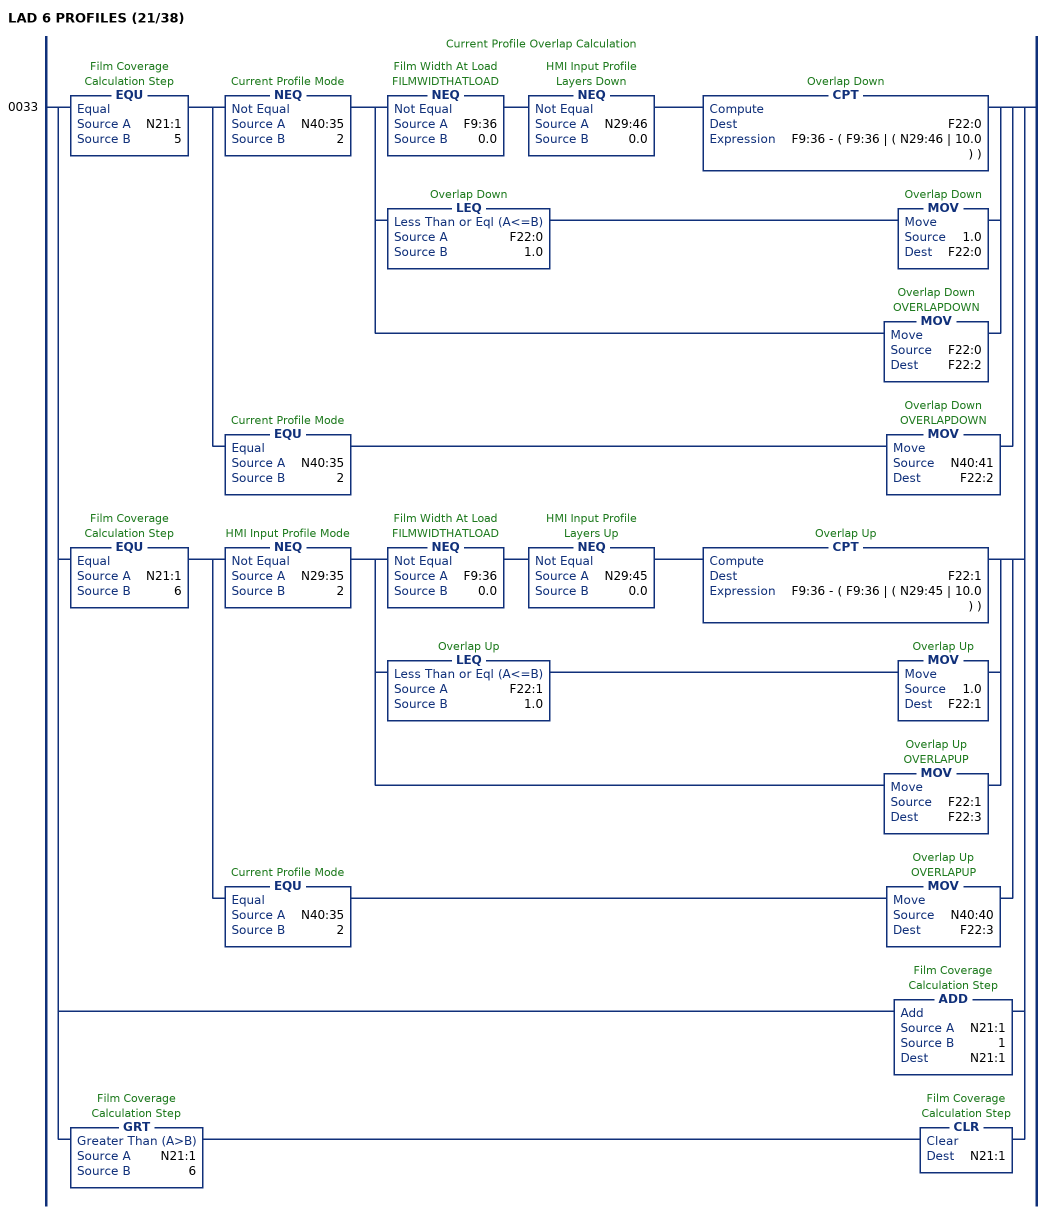
% Rung: 33 %
% Current Profile Overlap Calculation %
SOR BST EQU N21:1 5 BST NEQ N40:35 2 BST NEQ F9:36 0.0 NEQ N29:46 0.0 CPT F22:0 " F9:36 - ( F9:36 | ( N29:46 | 10.0 ) ) " NXB LEQ F22:0 1.0 MOV 1.0 F22:0 NXB MOV F22:0 F22:2 BND NXB EQU N40:35 2 MOV N40:41 F22:2 BND NXB EQU N21:1 6 BST NEQ N29:35 2 BST NEQ F9:36 0.0 NEQ N29:45 0.0 CPT F22:1 " F9:36 - ( F9:36 | ( N29:45 | 10.0 ) ) " NXB LEQ F22:1 1.0 MOV 1.0 F22:1 NXB MOV F22:1 F22:3 BND NXB EQU N40:35 2 MOV N40:40 F22:3 BND NXB BST ADD N21:1 1 N21:1 NXB GRT N21:1 6 CLR N21:1 BND BND EOR
%   N21:1  "Film Coverage Calculation Step" %
%   N40:35  "Current Profile Mode" %
%   F9:36  FILMWIDTHATLOAD  "Film Width At Load" %
%   N29:46  "HMI Input Profile Layers Down" %
%   F22:0  "Overlap Down" %
%   F22:2  OVERLAPDOWN  "Overlap Down" %
%   N29:35  "HMI Input Profile Mode" %
%   N29:45  "HMI Input Profile Layers Up" %
%   F22:1  "Overlap Up" %
%   F22:3  OVERLAPUP  "Overlap Up" %

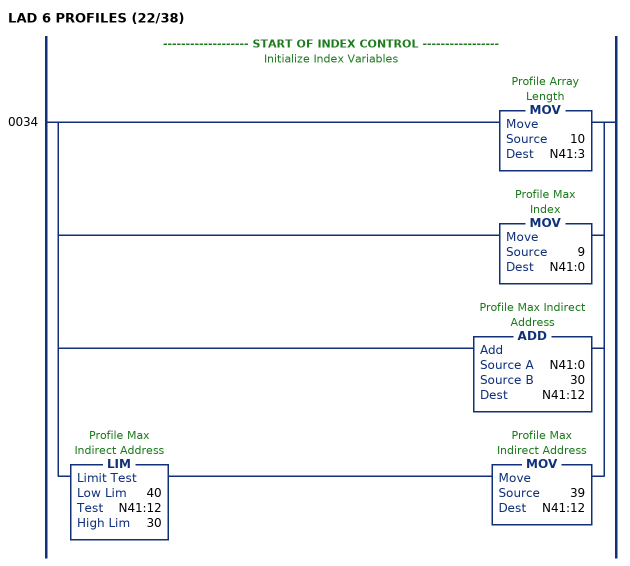
% Rung: 34 %
% TITLE: ------------------- START OF INDEX CONTROL ----------------- %
% Initialize Index Variables %
SOR BST MOV 10 N41:3 NXB MOV 9 N41:0 NXB ADD N41:0 30 N41:12 NXB LIM 40 N41:12 30 MOV 39 N41:12 BND EOR
%   N41:3  "Profile Array Length" %
%   N41:0  "Profile Max Index" %
%   N41:12  "Profile Max Indirect Address" %

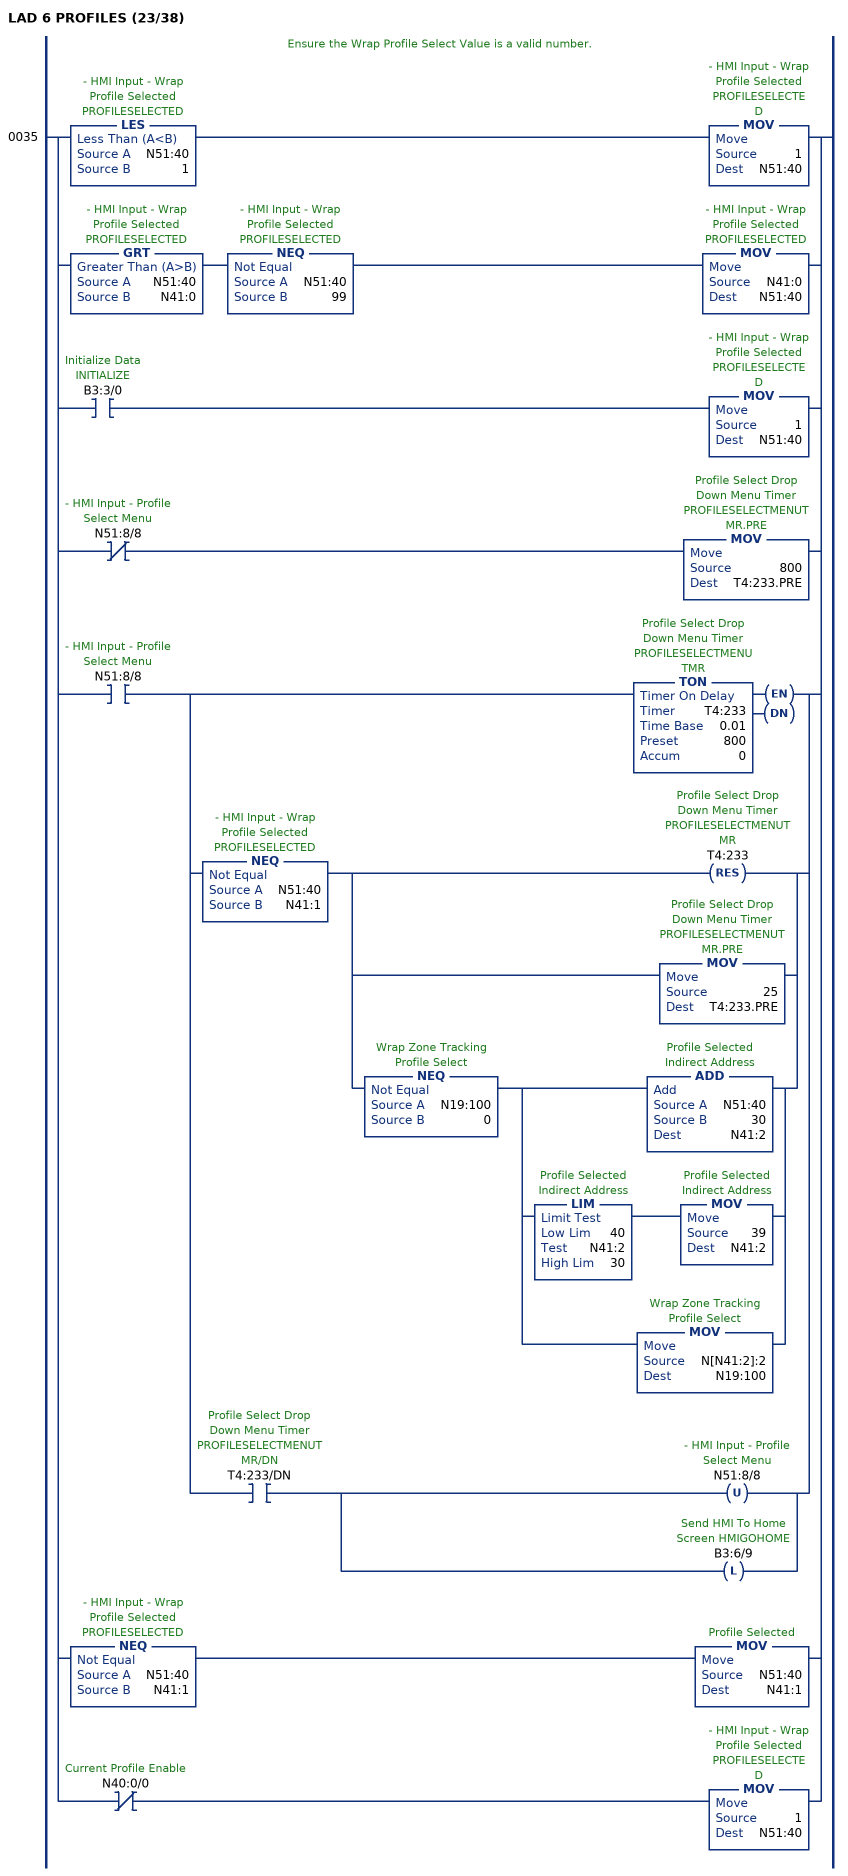
% Rung: 35 %
% Ensure the Wrap Profile Select Value is a valid number. %
SOR BST LES N51:40 1 MOV 1 N51:40 NXB GRT N51:40 N41:0 NEQ N51:40 99 MOV N41:0 N51:40 NXB XIC B3:3/0 MOV 1 N51:40 NXB XIO N51:8/8 MOV 800 T4:233.PRE NXB XIC N51:8/8 BST TON T4:233 0.01 800 0 NXB NEQ N51:40 N41:1 BST RES T4:233 NXB MOV 25 T4:233.PRE NXB NEQ N19:100 0 BST ADD N51:40 30 N41:2 NXB LIM 40 N41:2 30 MOV 39 N41:2 NXB MOV N[N41:2]:2 N19:100 BND BND NXB XIC T4:233/DN BST OTU N51:8/8 NXB OTL B3:6/9 BND BND NXB NEQ N51:40 N41:1 MOV N51:40 N41:1 NXB XIO N40:0/0 MOV 1 N51:40 BND EOR
%   N51:40  PROFILESELECTED  "- HMI Input - Wrap Profile Selected" %
%   N41:0  "Profile Max Index" %
%   B3:3/0  INITIALIZE  "Initialize Data" %
%   N51:8/8  "- HMI Input - Profile Select Menu" %
%   T4:233  PROFILESELECTMENUTMR  "Profile Select Drop Down Menu Timer" %
%   N41:1  "Profile Selected" %
%   N19:100  "Wrap Zone Tracking Profile Select" %
%   N41:2  "Profile Selected Indirect Address" %
%   B3:6/9  HMIGOHOME  "Send HMI To Home Screen" %
%   N40:0/0  "Current Profile Enable" %

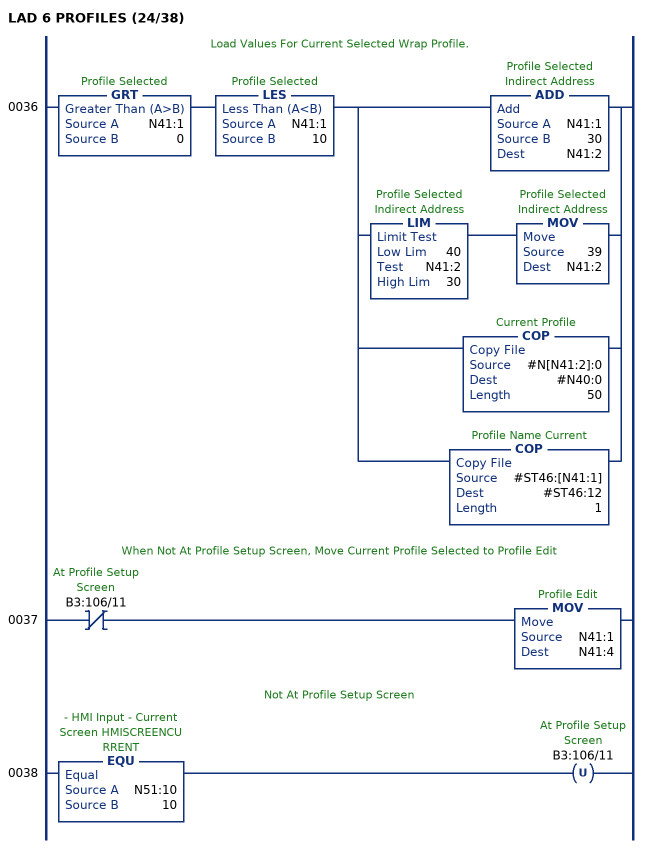
% Rung: 36 %
% Load Values For Current Selected Wrap Profile. %
SOR GRT N41:1 0 LES N41:1 10 BST ADD N41:1 30 N41:2 NXB LIM 40 N41:2 30 MOV 39 N41:2 NXB COP #N[N41:2]:0 #N40:0 50 NXB COP #ST46:[N41:1] #ST46:12 1 BND EOR
%   N41:1  "Profile Selected" %
%   N41:2  "Profile Selected Indirect Address" %
%   N40:0  "Current Profile" %
%   ST46:12  "Profile Name Current" %
% Rung: 37 %
% When Not At Profile Setup Screen, Move Current Profile Selected to Profile Edit %
SOR XIO B3:106/11 MOV N41:1 N41:4 EOR
%   B3:106/11  "At Profile Setup Screen" %
%   N41:1  "Profile Selected" %
%   N41:4  "Profile Edit" %
% Rung: 38 %
% Not At Profile Setup Screen %
SOR EQU N51:10 10 OTU B3:106/11 EOR
%   N51:10  HMISCREENCURRENT  "- HMI Input - Current Screen" %
%   B3:106/11  "At Profile Setup Screen" %

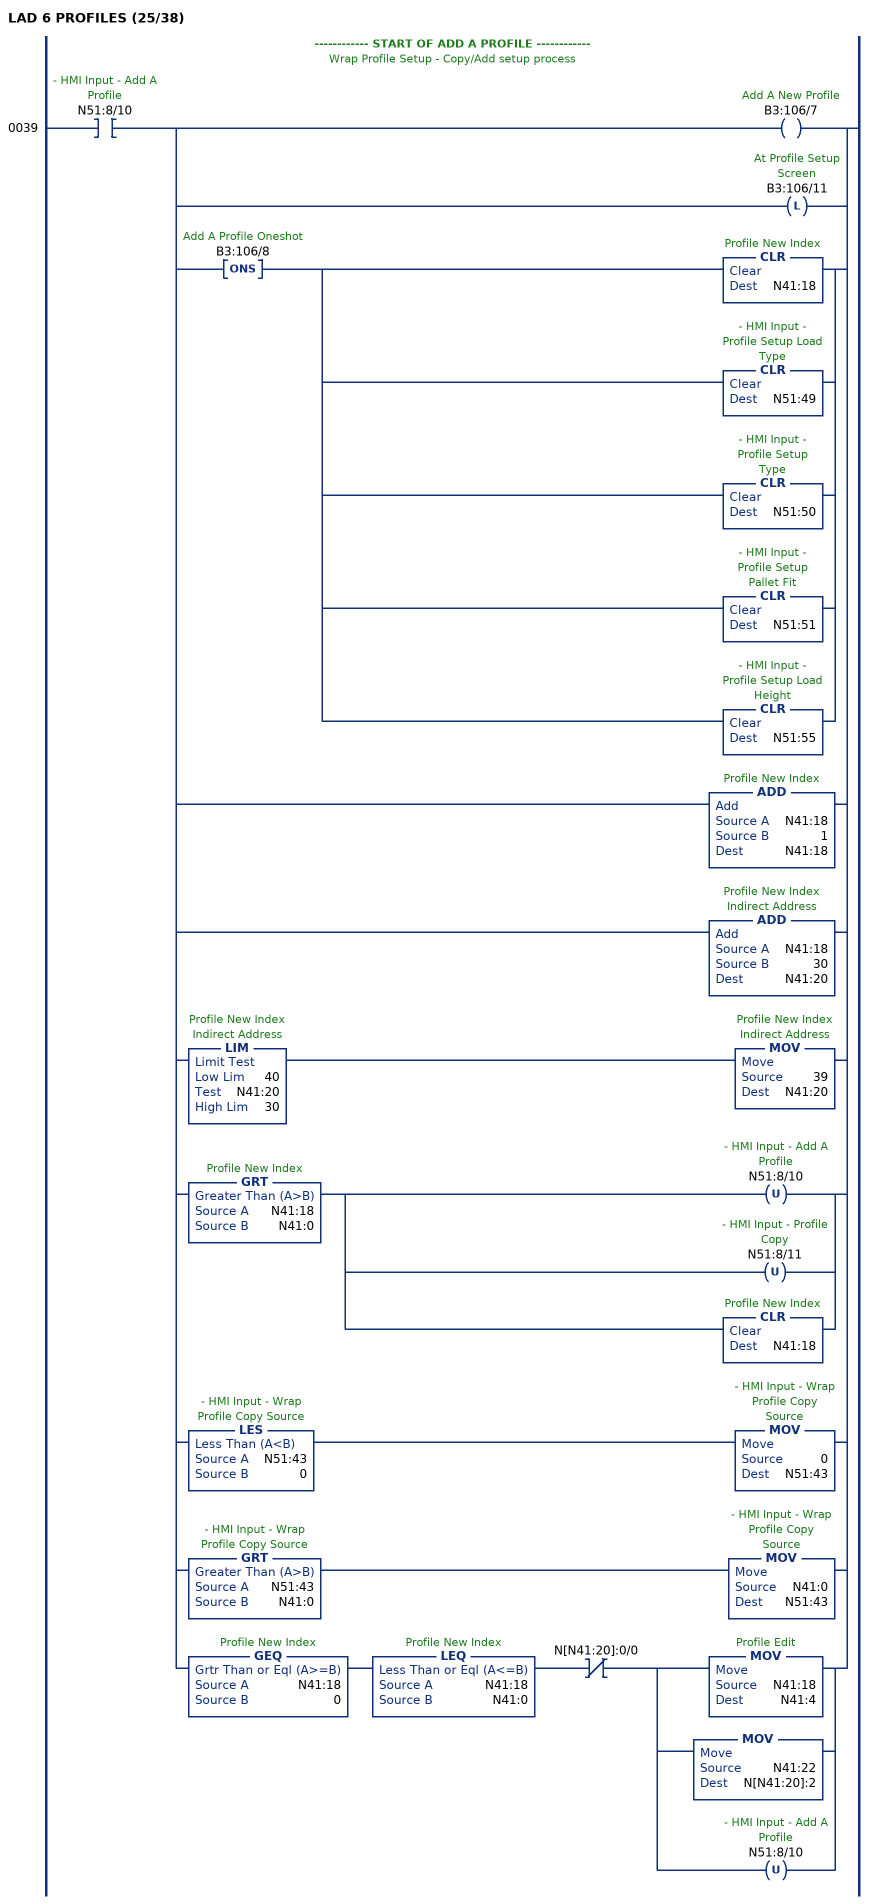
% Rung: 39 %
% TITLE: ------------ START OF ADD A PROFILE ------------ %
% Wrap Profile Setup - Copy/Add setup process %
SOR XIC N51:8/10 BST BST OTE B3:106/7 NXB OTL B3:106/11 BND NXB ONS B3:106/8 BST CLR N41:18 NXB CLR N51:49 NXB CLR N51:50 NXB CLR N51:51 NXB CLR N51:55 BND NXB BST ADD N41:18 1 N41:18 NXB ADD N41:18 30 N41:20 NXB LIM 40 N41:20 30 MOV 39 N41:20 BND NXB GRT N41:18 N41:0 BST OTU N51:8/10 NXB OTU N51:8/11 NXB CLR N41:18 BND NXB BST LES N51:43 0 MOV 0 N51:43 NXB GRT N51:43 N41:0 MOV N41:0 N51:43 BND NXB GEQ N41:18 0 LEQ N41:18 N41:0 XIO N[N41:20]:0/0 BST MOV N41:18 N41:4 NXB MOV N41:22 N[N41:20]:2 NXB OTU N51:8/10 BND BND EOR
%   N51:8/10  "- HMI Input - Add A Profile" %
%   B3:106/7  "Add A New Profile" %
%   B3:106/11  "At Profile Setup Screen" %
%   B3:106/8  "Add A Profile Oneshot" %
%   N41:18  "Profile New Index" %
%   N51:49  "- HMI Input - Profile Setup Load Type" %
%   N51:50  "- HMI Input - Profile Setup Type" %
%   N51:51  "- HMI Input - Profile Setup Pallet Fit" %
%   N51:55  "- HMI Input - Profile Setup Load Height" %
%   N41:20  "Profile New Index Indirect Address" %
%   N41:0  "Profile Max Index" %
%   N51:8/11  "- HMI Input - Profile Copy" %
%   N51:43  "- HMI Input - Wrap Profile Copy Source" %
%   N41:4  "Profile Edit" %
%   N41:22  "Profile Number Next" %

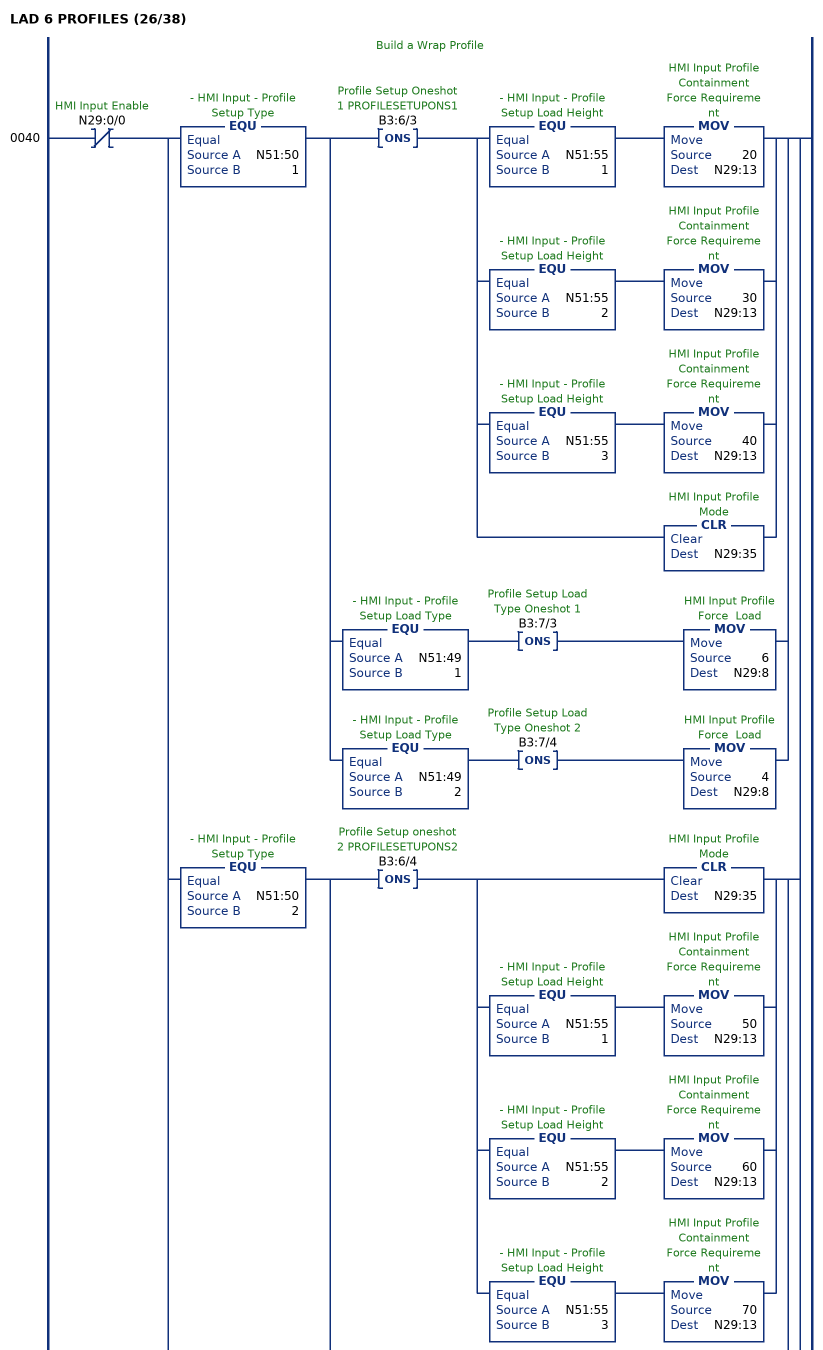

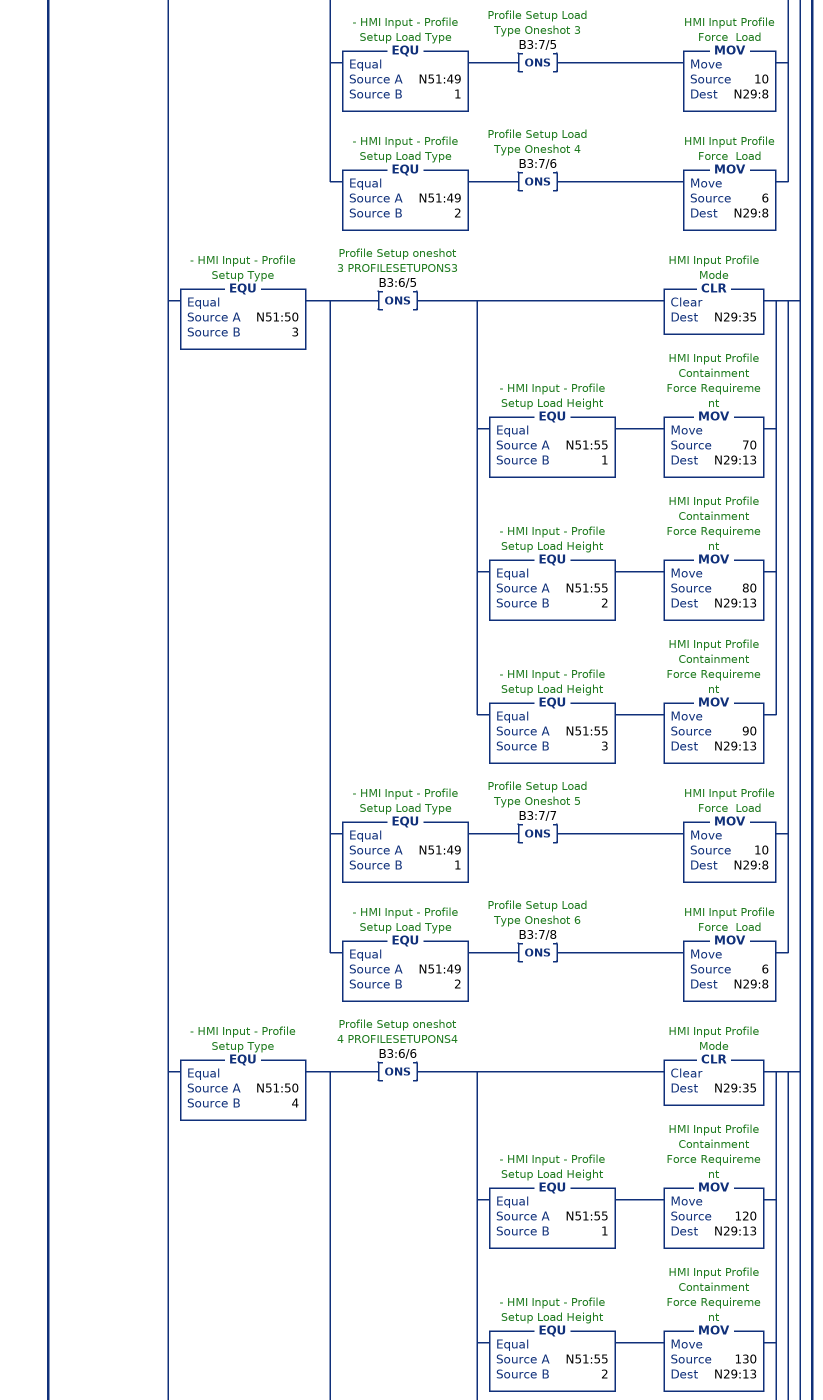

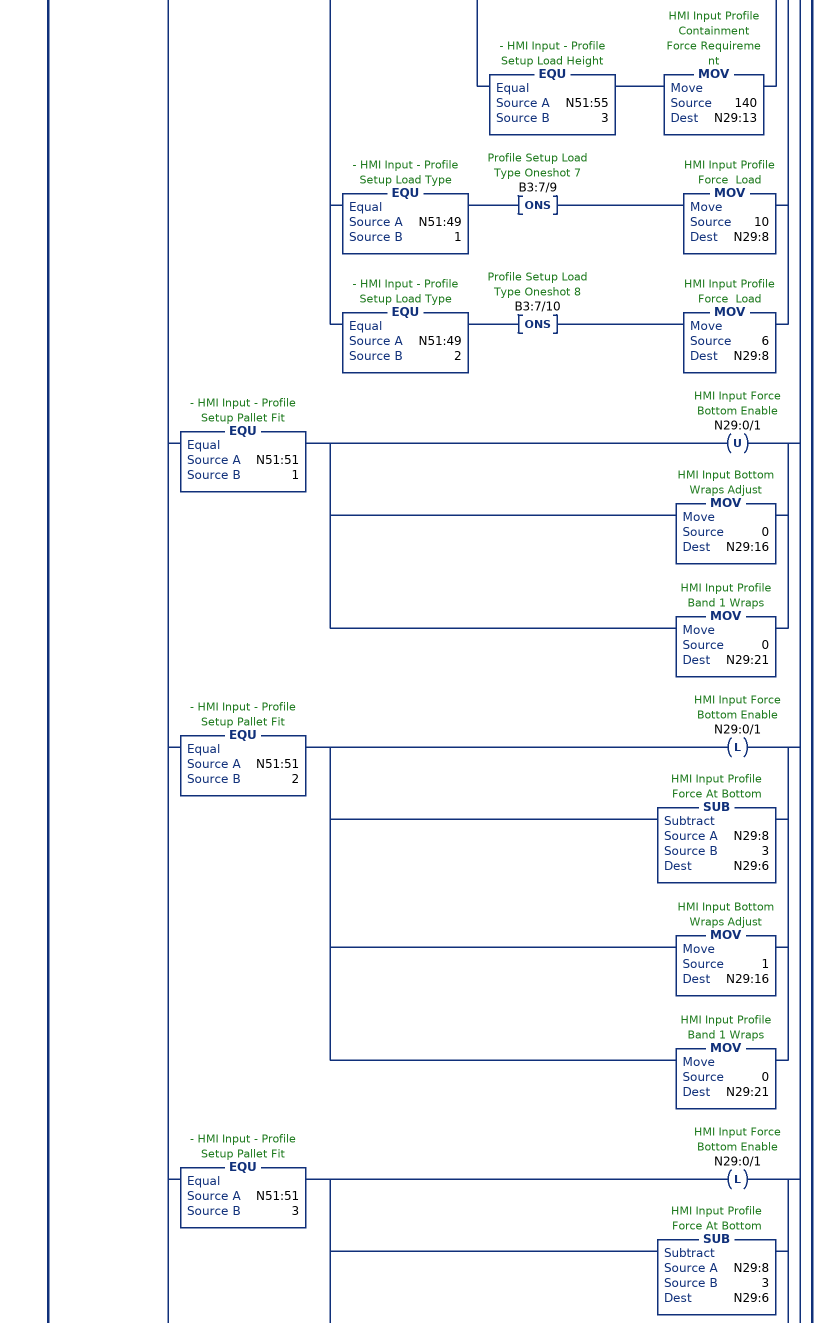

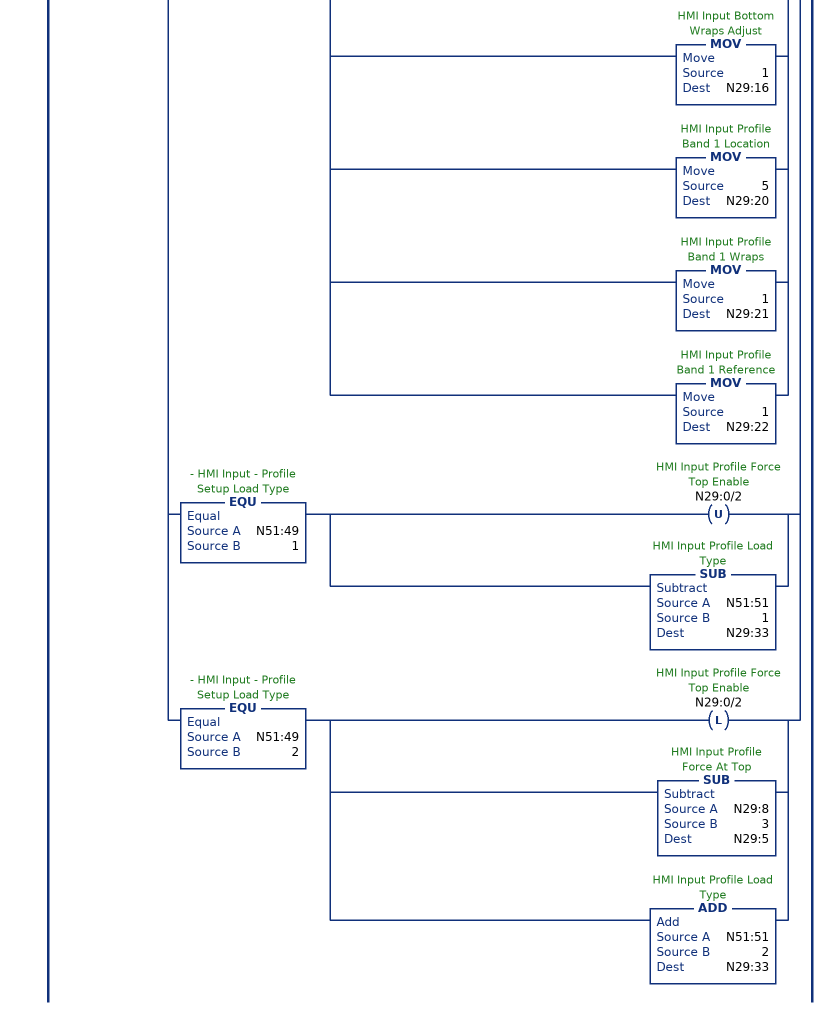
% Rung: 40 %
% Build a Wrap Profile %
SOR XIO N29:0/0 BST EQU N51:50 1 BST ONS B3:6/3 BST EQU N51:55 1 MOV 20 N29:13 NXB EQU N51:55 2 MOV 30 N29:13 NXB EQU N51:55 3 MOV 40 N29:13 NXB CLR N29:35 BND NXB BST EQU N51:49 1 ONS B3:7/3 MOV 6 N29:8 NXB EQU N51:49 2 ONS B3:7/4 MOV 4 N29:8 BND BND NXB EQU N51:50 2 BST ONS B3:6/4 BST CLR N29:35 NXB EQU N51:55 1 MOV 50 N29:13 NXB EQU N51:55 2 MOV 60 N29:13 NXB EQU N51:55 3 MOV 70 N29:13 BND NXB BST EQU N51:49 1 ONS B3:7/5 MOV 10 N29:8 NXB EQU N51:49 2 ONS B3:7/6 MOV 6 N29:8 BND BND NXB EQU N51:50 3 BST ONS B3:6/5 BST CLR N29:35 NXB EQU N51:55 1 MOV 70 N29:13 NXB EQU N51:55 2 MOV 80 N29:13 NXB EQU N51:55 3 MOV 90 N29:13 BND NXB BST EQU N51:49 1 ONS B3:7/7 MOV 10 N29:8 NXB EQU N51:49 2 ONS B3:7/8 MOV 6 N29:8 BND BND NXB EQU N51:50 4 BST ONS B3:6/6 BST CLR N29:35 NXB EQU N51:55 1 MOV 120 N29:13 NXB EQU N51:55 2 MOV 130 N29:13 NXB EQU N51:55 3 MOV 140 N29:13 BND NXB BST EQU N51:49 1 ONS B3:7/9 MOV 10 N29:8 NXB EQU N51:49 2 ONS B3:7/10 MOV 6 N29:8 BND BND NXB EQU N51:51 1 BST OTU N29:0/1 NXB MOV 0 N29:16 NXB MOV 0 N29:21 BND NXB EQU N51:51 2 BST OTL N29:0/1 NXB SUB N29:8 3 N29:6 NXB MOV 1 N29:16 NXB MOV 0 N29:21 BND NXB EQU N51:51 3 BST OTL N29:0/1 NXB SUB N29:8 3 N29:6 NXB MOV 1 N29:16 NXB MOV 5 N29:20 NXB MOV 1 N29:21 NXB MOV 1 N29:22 BND NXB EQU N51:49 1 BST OTU N29:0/2 NXB SUB N51:51 1 N29:33 BND NXB EQU N51:49 2 BST OTL N29:0/2 NXB SUB N29:8 3 N29:5 NXB ADD N51:51 2 N29:33 BND BND EOR
%   N29:0/0  "HMI Input Enable" %
%   N51:50  "- HMI Input - Profile Setup Type" %
%   B3:6/3  PROFILESETUPONS1  "Profile Setup Oneshot 1" %
%   N51:55  "- HMI Input - Profile Setup Load Height" %
%   N29:13  "HMI Input Profile Containment Force Requirement" %
%   N29:35  "HMI Input Profile Mode" %
%   N51:49  "- HMI Input - Profile Setup Load Type" %
%   B3:7/3  "Profile Setup Load Type Oneshot 1" %
%   N29:8  "HMI Input Profile Force  Load" %
%   B3:7/4  "Profile Setup Load Type Oneshot 2" %
%   B3:6/4  PROFILESETUPONS2  "Profile Setup oneshot 2" %
%   B3:7/5  "Profile Setup Load Type Oneshot 3" %
%   B3:7/6  "Profile Setup Load Type Oneshot 4" %
%   B3:6/5  PROFILESETUPONS3  "Profile Setup oneshot 3" %
%   B3:7/7  "Profile Setup Load Type Oneshot 5" %
%   B3:7/8  "Profile Setup Load Type Oneshot 6" %
%   B3:6/6  PROFILESETUPONS4  "Profile Setup oneshot 4" %
%   B3:7/9  "Profile Setup Load Type Oneshot 7" %
%   B3:7/10  "Profile Setup Load Type Oneshot 8" %
%   N51:51  "- HMI Input - Profile Setup Pallet Fit" %
%   N29:0/1  "HMI Input Force Bottom Enable" %
%   N29:16  "HMI Input Bottom Wraps Adjust" %
%   N29:21  "HMI Input Profile Band 1 Wraps" %
%   N29:6  "HMI Input Profile Force At Bottom" %
%   N29:20  "HMI Input Profile Band 1 Location" %
%   N29:22  "HMI Input Profile Band 1 Reference" %
%   N29:0/2  "HMI Input Profile Force Top Enable" %
%   N29:33  "HMI Input Profile Load Type" %
%   N29:5  "HMI Input Profile Force At Top" %

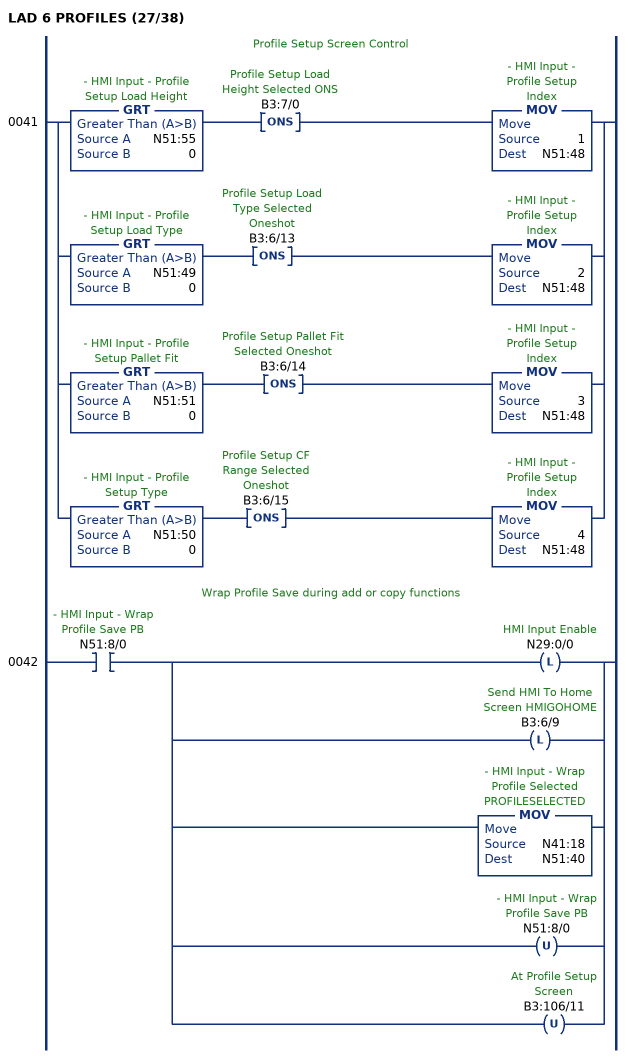
% Rung: 41 %
% Profile Setup Screen Control %
SOR BST GRT N51:55 0 ONS B3:7/0 MOV 1 N51:48 NXB GRT N51:49 0 ONS B3:6/13 MOV 2 N51:48 NXB GRT N51:51 0 ONS B3:6/14 MOV 3 N51:48 NXB GRT N51:50 0 ONS B3:6/15 MOV 4 N51:48 BND EOR
%   N51:55  "- HMI Input - Profile Setup Load Height" %
%   B3:7/0  "Profile Setup Load Height Selected ONS" %
%   N51:48  "- HMI Input - Profile Setup Index" %
%   N51:49  "- HMI Input - Profile Setup Load Type" %
%   B3:6/13  "Profile Setup Load Type Selected Oneshot" %
%   N51:51  "- HMI Input - Profile Setup Pallet Fit" %
%   B3:6/14  "Profile Setup Pallet Fit Selected Oneshot" %
%   N51:50  "- HMI Input - Profile Setup Type" %
%   B3:6/15  "Profile Setup CF Range Selected Oneshot" %
% Rung: 42 %
% Wrap Profile Save during add or copy functions %
SOR XIC N51:8/0 BST OTL N29:0/0 NXB OTL B3:6/9 NXB MOV N41:18 N51:40 NXB BST OTU N51:8/0 NXB OTU B3:106/11 BND BND EOR
%   N51:8/0  "- HMI Input - Wrap Profile Save PB" %
%   N29:0/0  "HMI Input Enable" %
%   B3:6/9  HMIGOHOME  "Send HMI To Home Screen" %
%   N41:18  "Profile New Index" %
%   N51:40  PROFILESELECTED  "- HMI Input - Wrap Profile Selected" %
%   B3:106/11  "At Profile Setup Screen" %

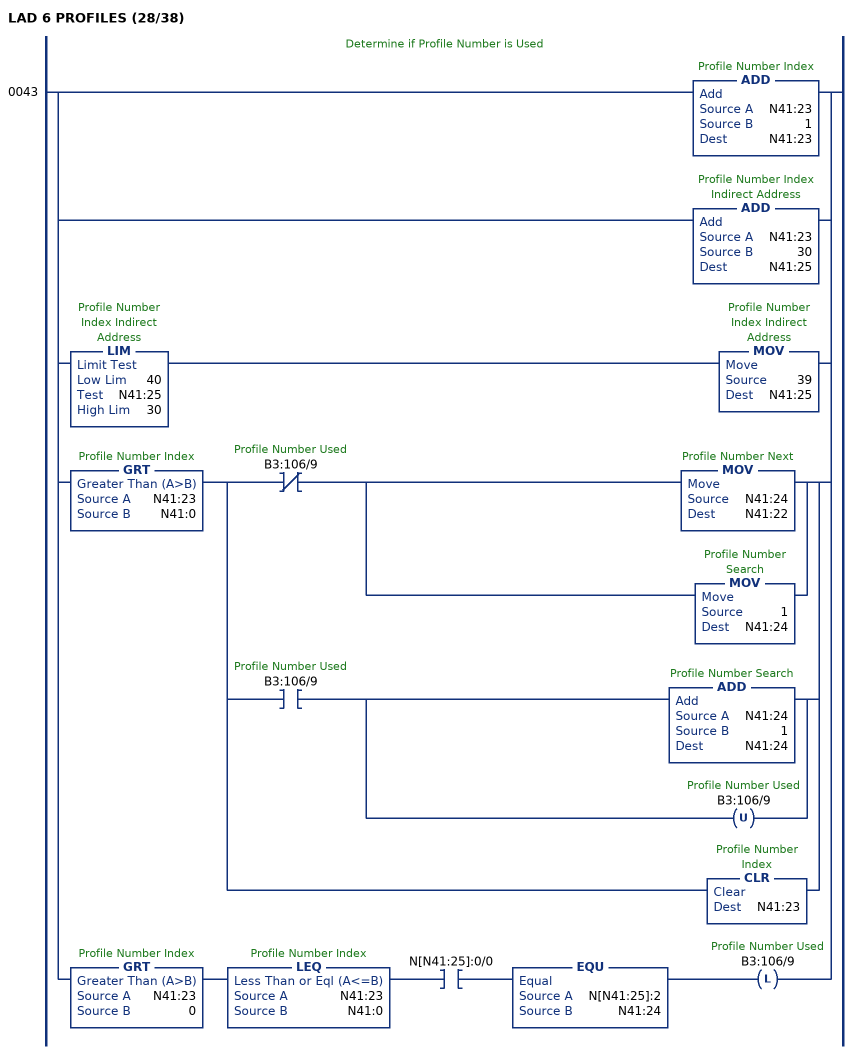
% Rung: 43 %
% Determine if Profile Number is Used %
SOR BST BST ADD N41:23 1 N41:23 NXB ADD N41:23 30 N41:25 NXB LIM 40 N41:25 30 MOV 39 N41:25 BND NXB GRT N41:23 N41:0 BST XIO B3:106/9 BST MOV N41:24 N41:22 NXB MOV 1 N41:24 BND NXB XIC B3:106/9 BST ADD N41:24 1 N41:24 NXB OTU B3:106/9 BND NXB CLR N41:23 BND NXB GRT N41:23 0 LEQ N41:23 N41:0 XIC N[N41:25]:0/0 EQU N[N41:25]:2 N41:24 OTL B3:106/9 BND EOR
%   N41:23  "Profile Number Index" %
%   N41:25  "Profile Number Index Indirect Address" %
%   N41:0  "Profile Max Index" %
%   B3:106/9  "Profile Number Used" %
%   N41:24  "Profile Number Search" %
%   N41:22  "Profile Number Next" %

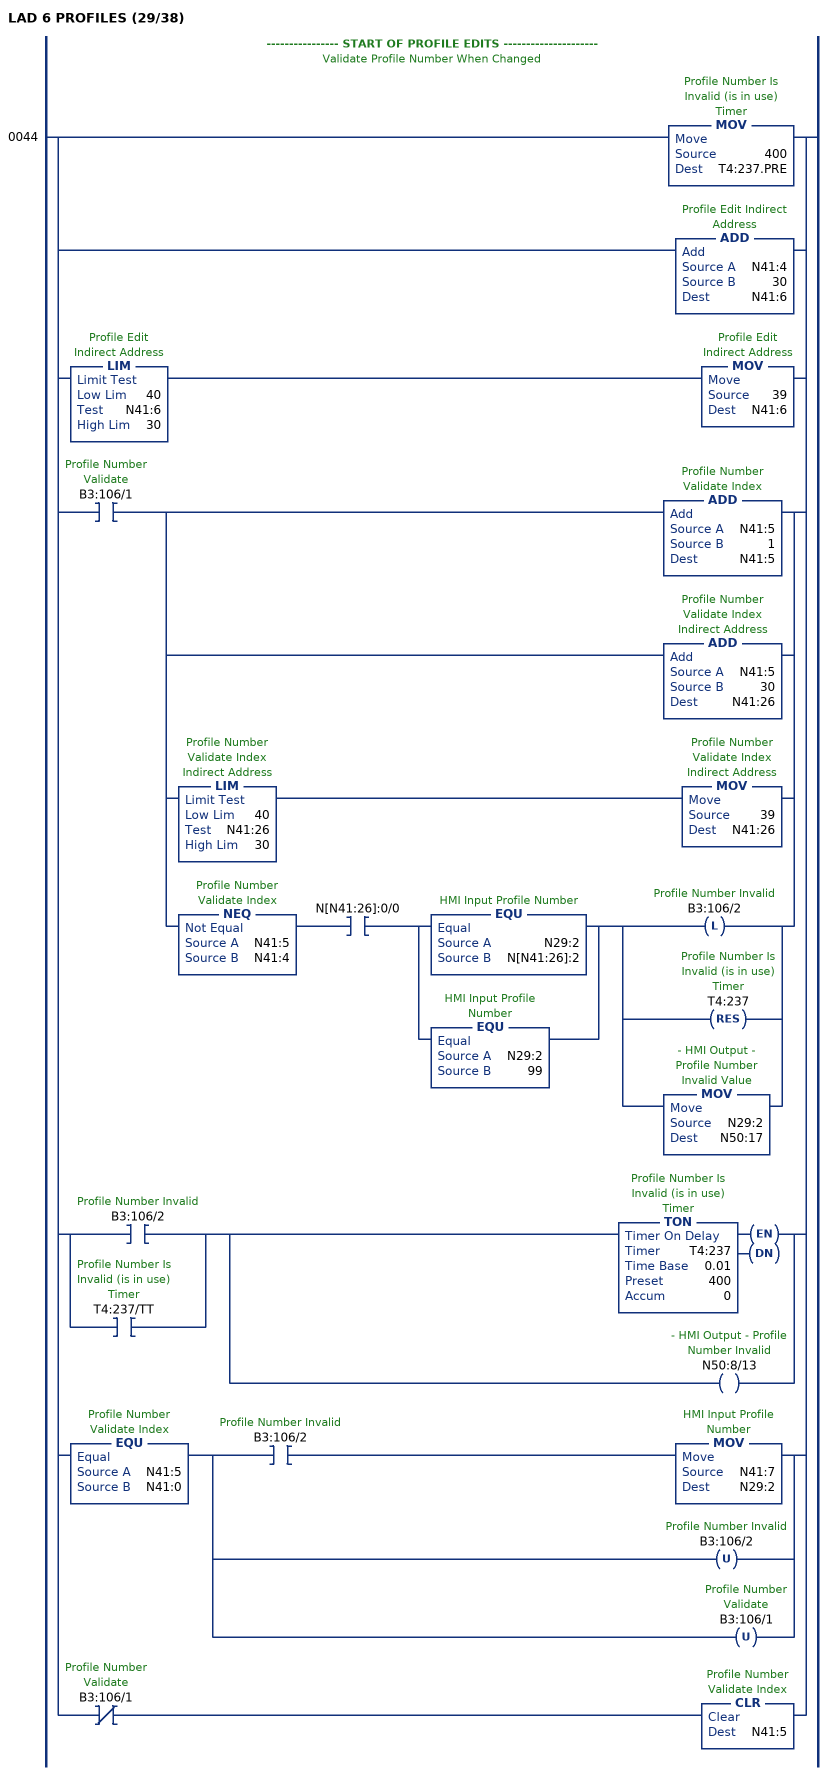
% Rung: 44 %
% TITLE: ---------------- START OF PROFILE EDITS --------------------- %
% Validate Profile Number When Changed %
SOR BST BST MOV 400 T4:237.PRE NXB ADD N41:4 30 N41:6 NXB LIM 40 N41:6 30 MOV 39 N41:6 BND NXB BST XIC B3:106/1 BST BST ADD N41:5 1 N41:5 NXB ADD N41:5 30 N41:26 NXB LIM 40 N41:26 30 MOV 39 N41:26 BND NXB NEQ N41:5 N41:4 XIC N[N41:26]:0/0 BST EQU N29:2 N[N41:26]:2 NXB EQU N29:2 99 BND BST OTL B3:106/2 NXB RES T4:237 NXB MOV N29:2 N50:17 BND BND NXB BST XIC B3:106/2 NXB XIC T4:237/TT BND BST TON T4:237 0.01 400 0 NXB OTE N50:8/13 BND NXB EQU N41:5 N41:0 BST XIC B3:106/2 MOV N41:7 N29:2 NXB OTU B3:106/2 NXB OTU B3:106/1 BND NXB XIO B3:106/1 CLR N41:5 BND BND EOR
%   T4:237  "Profile Number Is Invalid (is in use) Timer" %
%   N41:4  "Profile Edit" %
%   N41:6  "Profile Edit Indirect Address" %
%   B3:106/1  "Profile Number Validate" %
%   N41:5  "Profile Number Validate Index" %
%   N41:26  "Profile Number Validate Index Indirect Address" %
%   N29:2  "HMI Input Profile Number" %
%   B3:106/2  "Profile Number Invalid" %
%   N50:17  "- HMI Output - Profile Number Invalid Value" %
%   N50:8/13  "- HMI Output - Profile Number Invalid" %
%   N41:0  "Profile Max Index" %
%   N41:7  "Profile Number Check" %

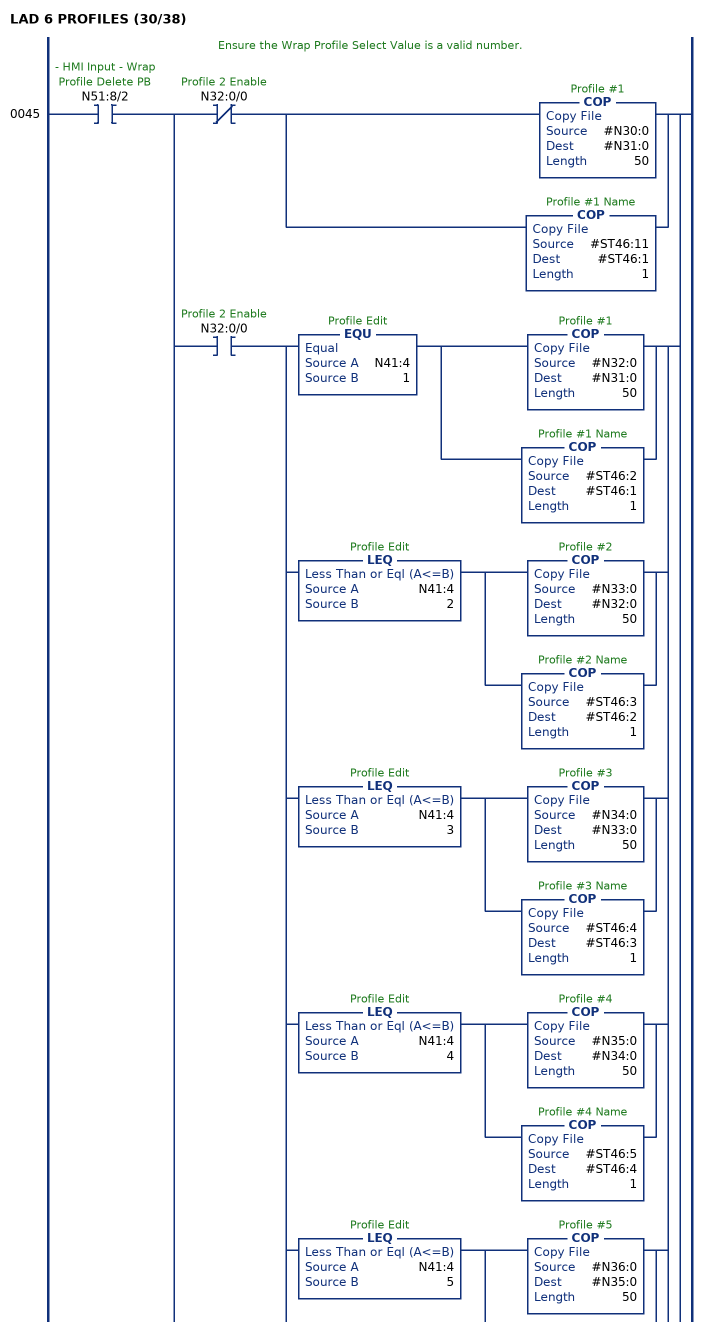

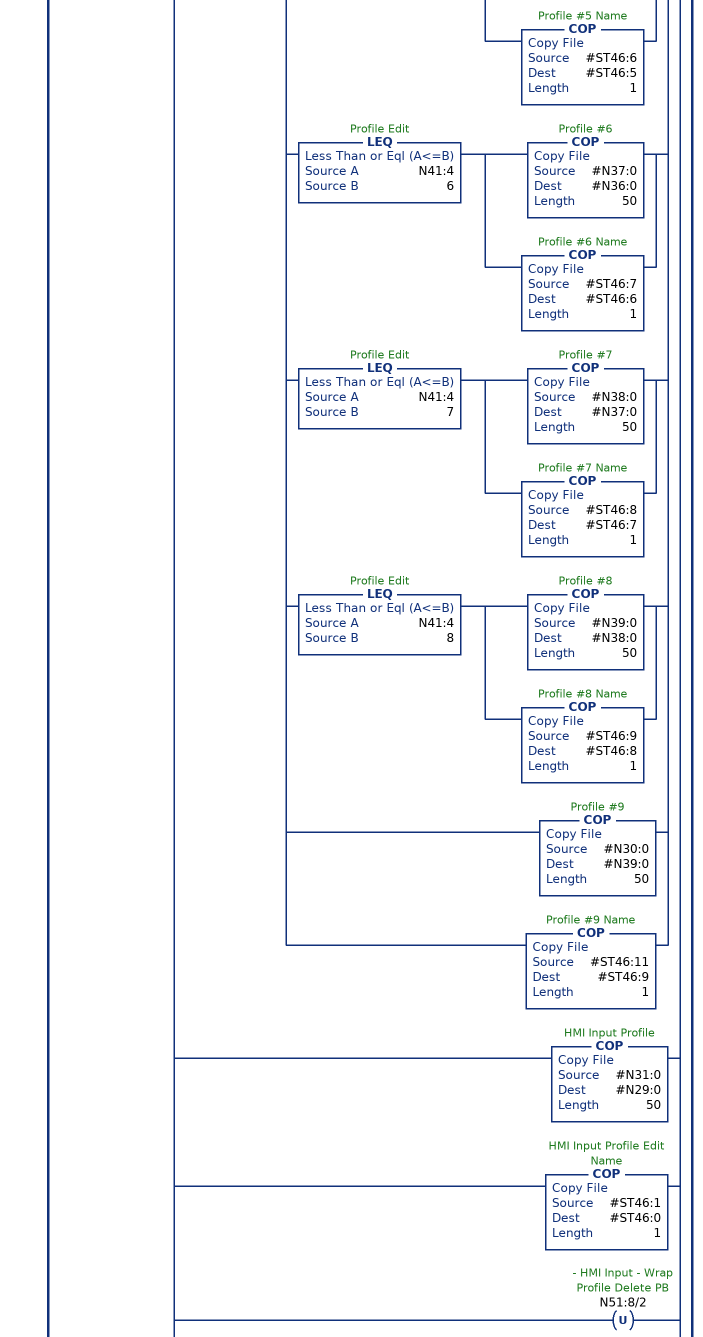

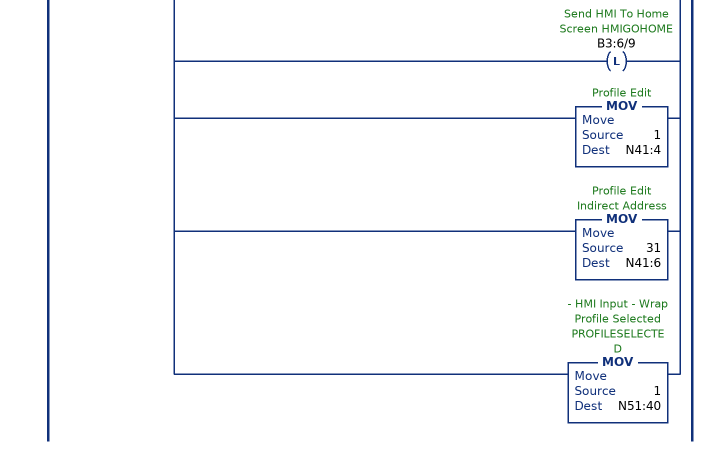
% Rung: 45 %
% Ensure the Wrap Profile Select Value is a valid number. %
SOR XIC N51:8/2 BST XIO N32:0/0 BST COP #N30:0 #N31:0 50 NXB COP #ST46:11 #ST46:1 1 BND NXB XIC N32:0/0 BST EQU N41:4 1 BST COP #N32:0 #N31:0 50 NXB COP #ST46:2 #ST46:1 1 BND NXB LEQ N41:4 2 BST COP #N33:0 #N32:0 50 NXB COP #ST46:3 #ST46:2 1 BND NXB LEQ N41:4 3 BST COP #N34:0 #N33:0 50 NXB COP #ST46:4 #ST46:3 1 BND NXB LEQ N41:4 4 BST COP #N35:0 #N34:0 50 NXB COP #ST46:5 #ST46:4 1 BND NXB LEQ N41:4 5 BST COP #N36:0 #N35:0 50 NXB COP #ST46:6 #ST46:5 1 BND NXB LEQ N41:4 6 BST COP #N37:0 #N36:0 50 NXB COP #ST46:7 #ST46:6 1 BND NXB LEQ N41:4 7 BST COP #N38:0 #N37:0 50 NXB COP #ST46:8 #ST46:7 1 BND NXB LEQ N41:4 8 BST COP #N39:0 #N38:0 50 NXB COP #ST46:9 #ST46:8 1 BND NXB BST COP #N30:0 #N39:0 50 NXB COP #ST46:11 #ST46:9 1 BND BND NXB BST COP #N31:0 #N29:0 50 NXB COP #ST46:1 #ST46:0 1 NXB OTU N51:8/2 NXB OTL B3:6/9 NXB MOV 1 N41:4 NXB MOV 31 N41:6 NXB MOV 1 N51:40 BND BND EOR
%   N51:8/2  "- HMI Input - Wrap Profile Delete PB" %
%   N32:0/0  "Profile 2 Enable" %
%   N30:0  "Enable bits" %
%   N31:0  "Profile #1" %
%   ST46:11  NULLSTRING  "Default Name For "Make a Copy" Profile" %
%   ST46:1  "Profile #1 Name" %
%   N41:4  "Profile Edit" %
%   N32:0  "Profile #2" %
%   ST46:2  "Profile #2 Name" %
%   N33:0  "Profile #3" %
%   ST46:3  "Profile #3 Name" %
%   N34:0  "Profile #4" %
%   ST46:4  "Profile #4 Name" %
%   N35:0  "Profile #5" %
%   ST46:5  "Profile #5 Name" %
%   N36:0  "Profile #6" %
%   ST46:6  "Profile #6 Name" %
%   N37:0  "Profile #7" %
%   ST46:7  "Profile #7 Name" %
%   N38:0  "Profile #8" %
%   ST46:8  "Profile #8 Name" %
%   N39:0  "Profile #9" %
%   ST46:9  "Profile #9 Name" %
%   N29:0  "HMI Input Profile" %
%   ST46:0  "HMI Input Profile Edit Name" %
%   B3:6/9  HMIGOHOME  "Send HMI To Home Screen" %
%   N41:6  "Profile Edit Indirect Address" %
%   N51:40  PROFILESELECTED  "- HMI Input - Wrap Profile Selected" %

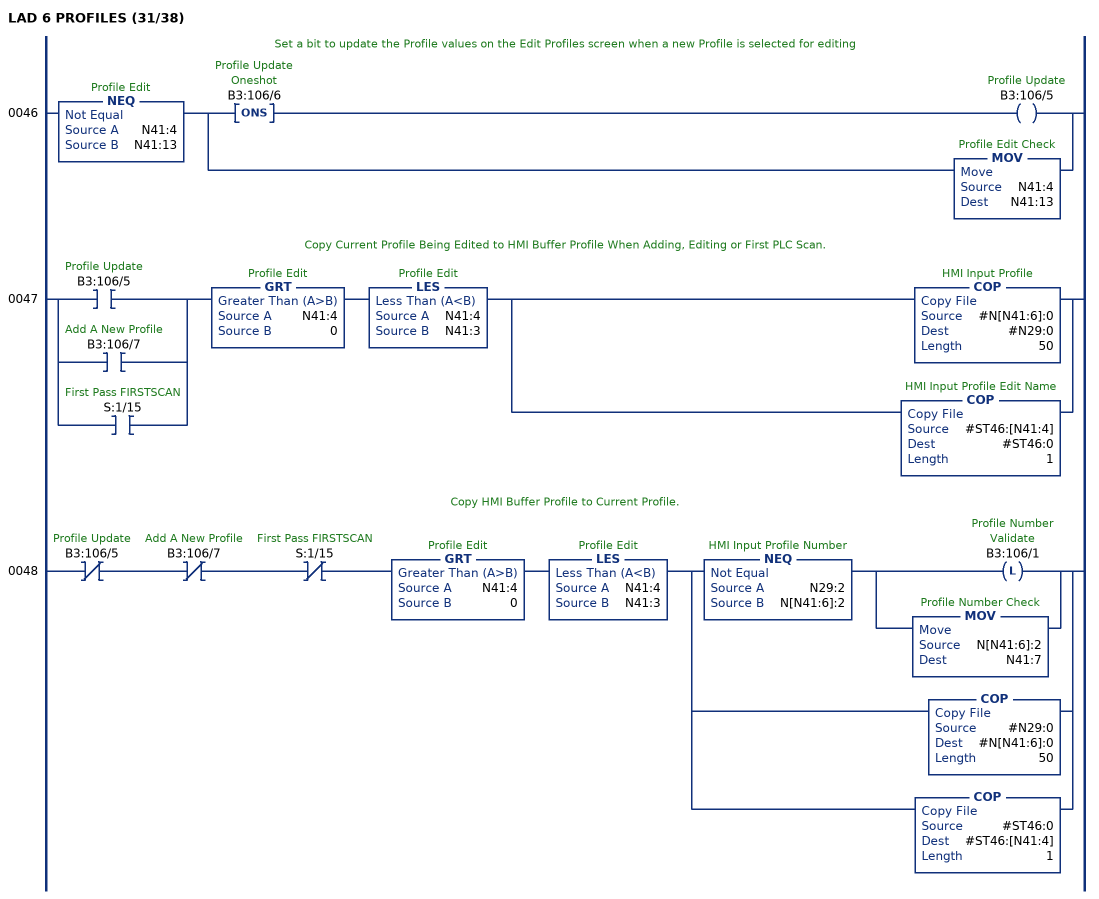
% Rung: 46 %
% Set a bit to update the Profile values on the Edit Profiles screen when a new Profile is selected for editing %
SOR NEQ N41:4 N41:13 BST ONS B3:106/6 OTE B3:106/5 NXB MOV N41:4 N41:13 BND EOR
%   N41:4  "Profile Edit" %
%   N41:13  "Profile Edit Check" %
%   B3:106/6  "Profile Update Oneshot" %
%   B3:106/5  "Profile Update" %
% Rung: 47 %
% Copy Current Profile Being Edited to HMI Buffer Profile When Adding, Editing or First PLC Scan. %
SOR BST XIC B3:106/5 NXB XIC B3:106/7 NXB XIC S:1/15 BND GRT N41:4 0 LES N41:4 N41:3 BST COP #N[N41:6]:0 #N29:0 50 NXB COP #ST46:[N41:4] #ST46:0 1 BND EOR
%   B3:106/5  "Profile Update" %
%   B3:106/7  "Add A New Profile" %
%   S:1/15  FIRSTSCAN  "First Pass" %
%   N41:4  "Profile Edit" %
%   N41:3  "Profile Array Length" %
%   N41:6  "Profile Edit Indirect Address" %
%   N29:0  "HMI Input Profile" %
%   ST46:0  "HMI Input Profile Edit Name" %
% Rung: 48 %
% Copy HMI Buffer Profile to Current Profile. %
SOR XIO B3:106/5 XIO B3:106/7 XIO S:1/15 GRT N41:4 0 LES N41:4 N41:3 BST NEQ N29:2 N[N41:6]:2 BST OTL B3:106/1 NXB MOV N[N41:6]:2 N41:7 BND NXB BST COP #N29:0 #N[N41:6]:0 50 NXB COP #ST46:0 #ST46:[N41:4] 1 BND BND EOR
%   B3:106/5  "Profile Update" %
%   B3:106/7  "Add A New Profile" %
%   S:1/15  FIRSTSCAN  "First Pass" %
%   N41:4  "Profile Edit" %
%   N41:3  "Profile Array Length" %
%   N29:2  "HMI Input Profile Number" %
%   N41:6  "Profile Edit Indirect Address" %
%   B3:106/1  "Profile Number Validate" %
%   N41:7  "Profile Number Check" %
%   N29:0  "HMI Input Profile" %
%   ST46:0  "HMI Input Profile Edit Name" %

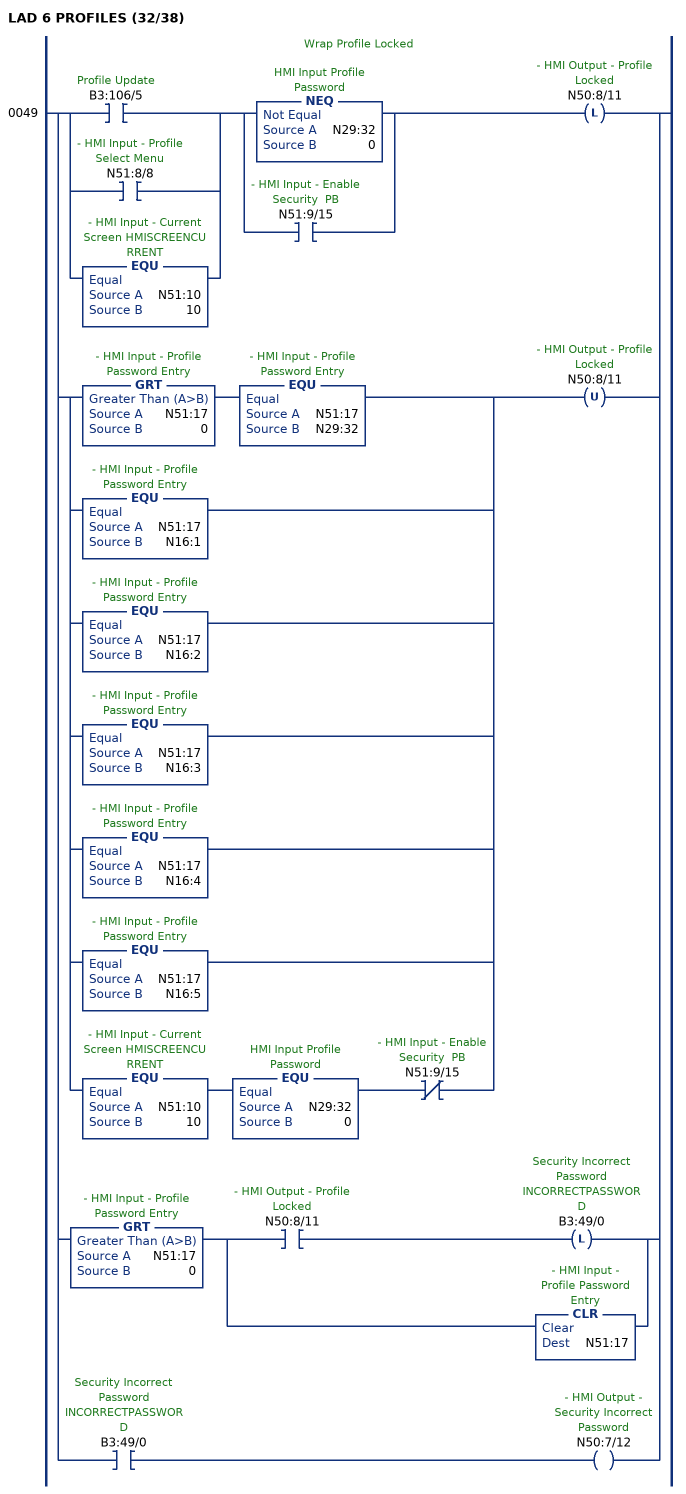
% Rung: 49 %
% Wrap Profile Locked %
SOR BST BST XIC B3:106/5 NXB XIC N51:8/8 NXB EQU N51:10 10 BND BST NEQ N29:32 0 NXB XIC N51:9/15 BND OTL N50:8/11 NXB BST GRT N51:17 0 EQU N51:17 N29:32 NXB EQU N51:17 N16:1 NXB EQU N51:17 N16:2 NXB EQU N51:17 N16:3 NXB EQU N51:17 N16:4 NXB EQU N51:17 N16:5 NXB EQU N51:10 10 EQU N29:32 0 XIO N51:9/15 BND OTU N50:8/11 NXB GRT N51:17 0 BST XIC N50:8/11 OTL B3:49/0 NXB CLR N51:17 BND NXB XIC B3:49/0 OTE N50:7/12 BND EOR
%   B3:106/5  "Profile Update" %
%   N51:8/8  "- HMI Input - Profile Select Menu" %
%   N51:10  HMISCREENCURRENT  "- HMI Input - Current Screen" %
%   N29:32  "HMI Input Profile Password" %
%   N51:9/15  "- HMI Input - Enable Security  PB" %
%   N50:8/11  "- HMI Output - Profile Locked" %
%   N51:17  "- HMI Input - Profile Password Entry" %
%   N16:1  "Level 1 Password" %
%   N16:2  "Level 2 Password" %
%   N16:3  "Lantech Password" %
%   N16:4  "Lantech Password" %
%   N16:5  "Lantech Password" %
%   B3:49/0  INCORRECTPASSWORD  "Security Incorrect Password" %
%   N50:7/12  "- HMI Output - Security Incorrect Password" %

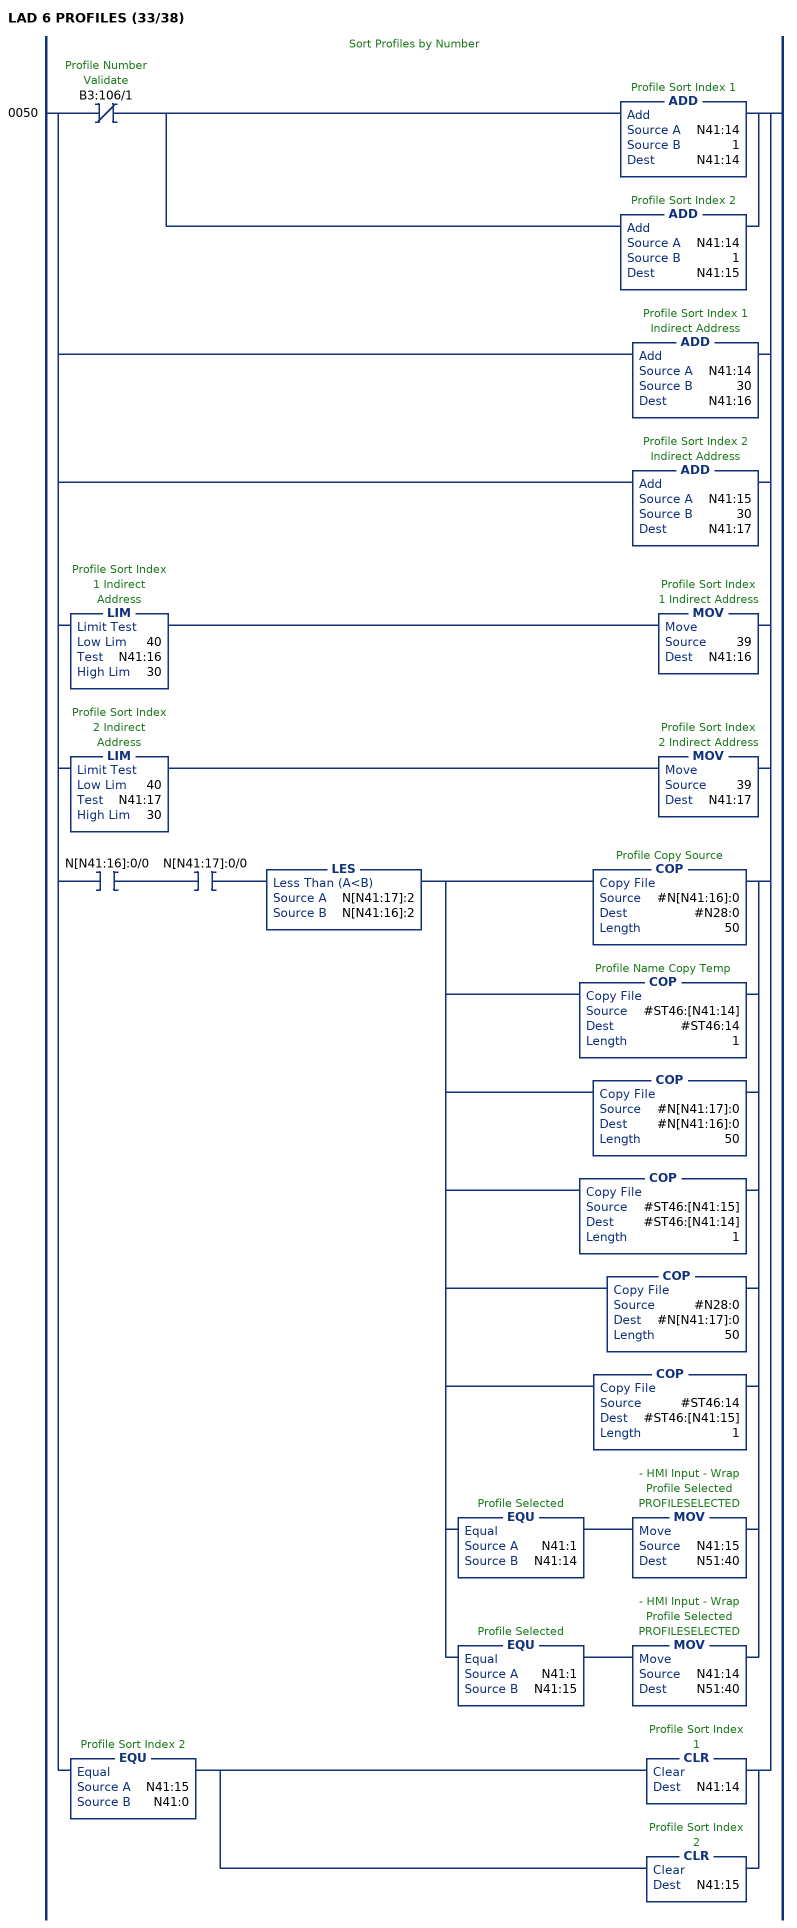
% Rung: 50 %
% Sort Profiles by Number %
SOR BST XIO B3:106/1 BST ADD N41:14 1 N41:14 NXB ADD N41:14 1 N41:15 BND NXB BST ADD N41:14 30 N41:16 NXB ADD N41:15 30 N41:17 NXB LIM 40 N41:16 30 MOV 39 N41:16 NXB LIM 40 N41:17 30 MOV 39 N41:17 BND NXB XIC N[N41:16]:0/0 XIC N[N41:17]:0/0 LES N[N41:17]:2 N[N41:16]:2 BST BST COP #N[N41:16]:0 #N28:0 50 NXB COP #ST46:[N41:14] #ST46:14 1 BND NXB BST COP #N[N41:17]:0 #N[N41:16]:0 50 NXB COP #ST46:[N41:15] #ST46:[N41:14] 1 BND NXB BST COP #N28:0 #N[N41:17]:0 50 NXB COP #ST46:14 #ST46:[N41:15] 1 BND NXB EQU N41:1 N41:14 MOV N41:15 N51:40 NXB EQU N41:1 N41:15 MOV N41:14 N51:40 BND NXB EQU N41:15 N41:0 BST CLR N41:14 NXB CLR N41:15 BND BND EOR
%   B3:106/1  "Profile Number Validate" %
%   N41:14  "Profile Sort Index 1" %
%   N41:15  "Profile Sort Index 2" %
%   N41:16  "Profile Sort Index 1 Indirect Address" %
%   N41:17  "Profile Sort Index 2 Indirect Address" %
%   N28:0  "Profile Copy Source" %
%   ST46:14  "Profile Name Copy Temp" %
%   N41:1  "Profile Selected" %
%   N51:40  PROFILESELECTED  "- HMI Input - Wrap Profile Selected" %
%   N41:0  "Profile Max Index" %

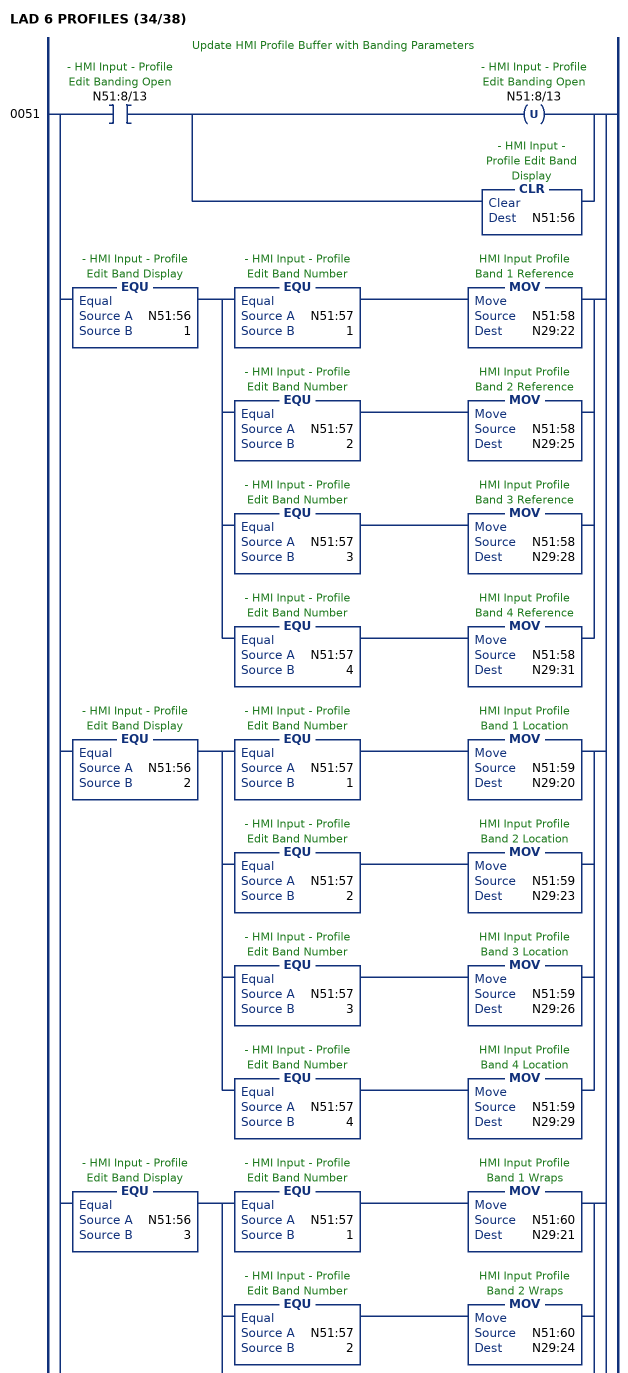

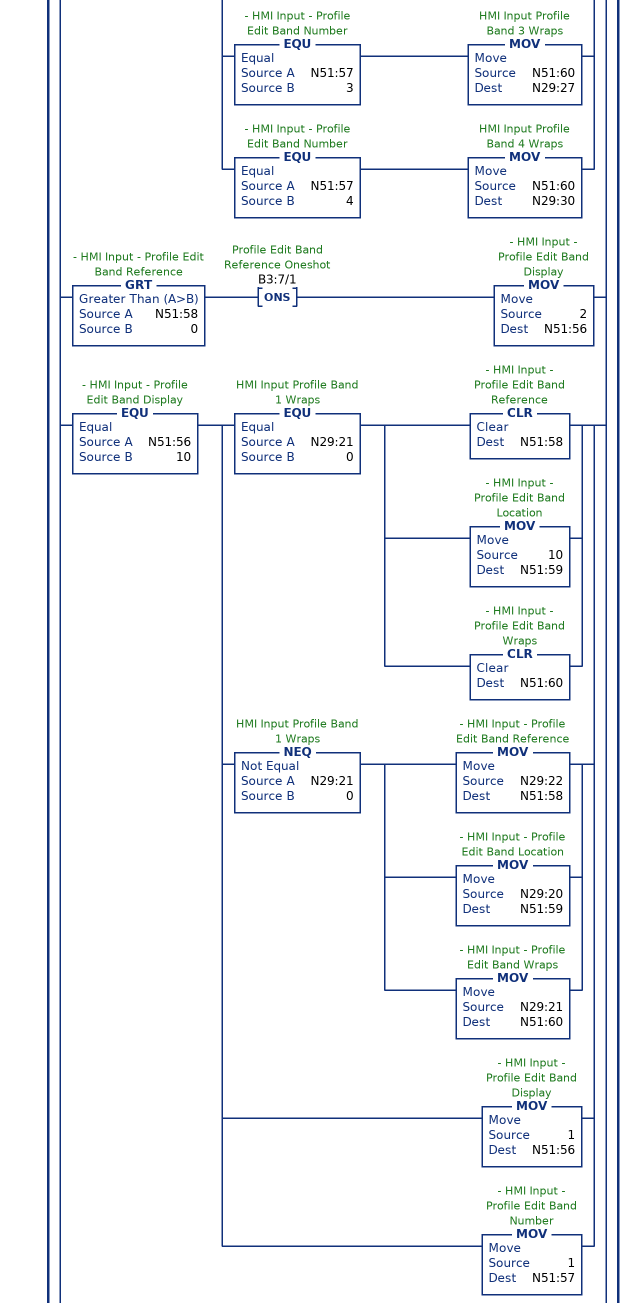

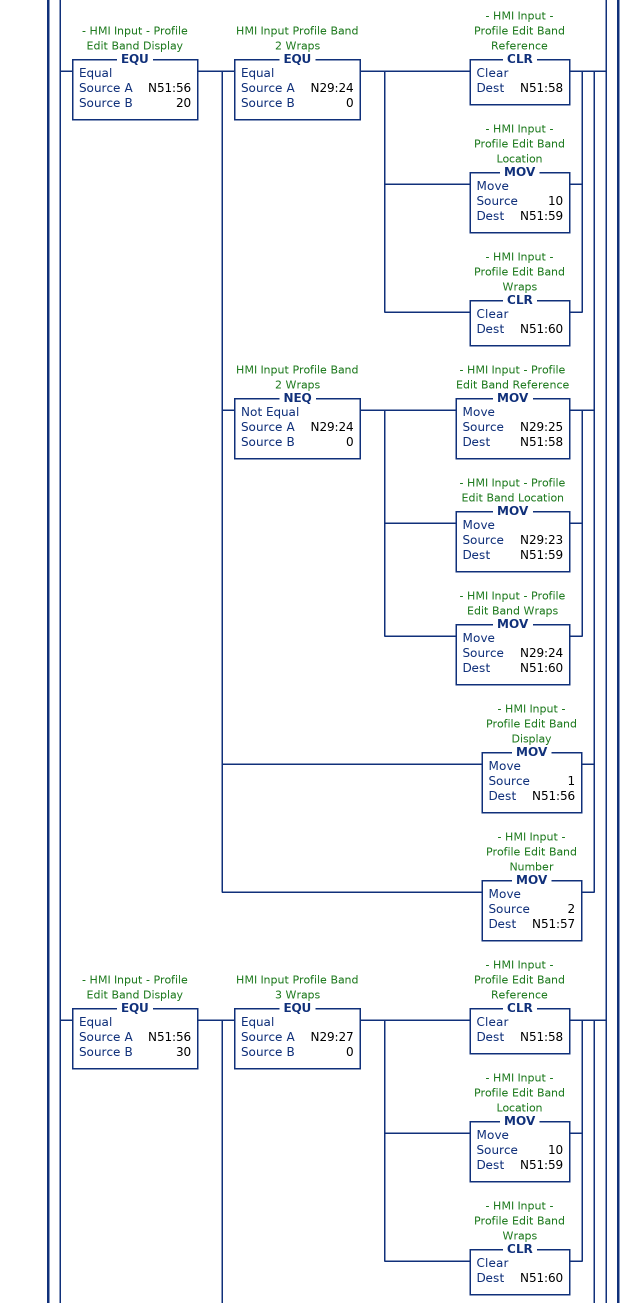

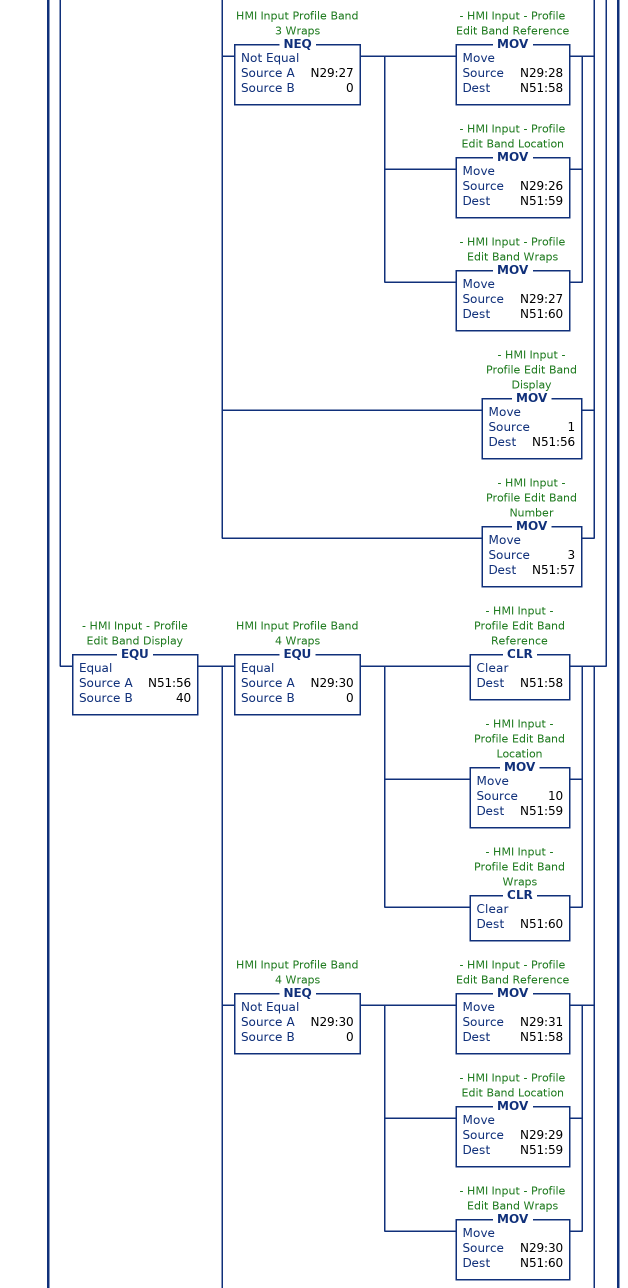

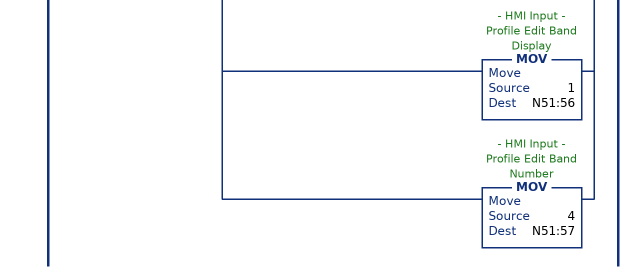
% Rung: 51 %
% Update HMI Profile Buffer with Banding Parameters %
SOR BST XIC N51:8/13 BST OTU N51:8/13 NXB CLR N51:56 BND NXB EQU N51:56 1 BST EQU N51:57 1 MOV N51:58 N29:22 NXB EQU N51:57 2 MOV N51:58 N29:25 NXB EQU N51:57 3 MOV N51:58 N29:28 NXB EQU N51:57 4 MOV N51:58 N29:31 BND NXB EQU N51:56 2 BST EQU N51:57 1 MOV N51:59 N29:20 NXB EQU N51:57 2 MOV N51:59 N29:23 NXB EQU N51:57 3 MOV N51:59 N29:26 NXB EQU N51:57 4 MOV N51:59 N29:29 BND NXB EQU N51:56 3 BST EQU N51:57 1 MOV N51:60 N29:21 NXB EQU N51:57 2 MOV N51:60 N29:24 NXB EQU N51:57 3 MOV N51:60 N29:27 NXB EQU N51:57 4 MOV N51:60 N29:30 BND NXB GRT N51:58 0 ONS B3:7/1 MOV 2 N51:56 NXB EQU N51:56 10 BST EQU N29:21 0 BST CLR N51:58 NXB MOV 10 N51:59 NXB CLR N51:60 BND NXB NEQ N29:21 0 BST MOV N29:22 N51:58 NXB MOV N29:20 N51:59 NXB MOV N29:21 N51:60 BND NXB MOV 1 N51:56 NXB MOV 1 N51:57 BND NXB EQU N51:56 20 BST EQU N29:24 0 BST CLR N51:58 NXB MOV 10 N51:59 NXB CLR N51:60 BND NXB NEQ N29:24 0 BST MOV N29:25 N51:58 NXB MOV N29:23 N51:59 NXB MOV N29:24 N51:60 BND NXB MOV 1 N51:56 NXB MOV 2 N51:57 BND NXB EQU N51:56 30 BST EQU N29:27 0 BST CLR N51:58 NXB MOV 10 N51:59 NXB CLR N51:60 BND NXB NEQ N29:27 0 BST MOV N29:28 N51:58 NXB MOV N29:26 N51:59 NXB MOV N29:27 N51:60 BND NXB MOV 1 N51:56 NXB MOV 3 N51:57 BND NXB EQU N51:56 40 BST EQU N29:30 0 BST CLR N51:58 NXB MOV 10 N51:59 NXB CLR N51:60 BND NXB NEQ N29:30 0 BST MOV N29:31 N51:58 NXB MOV N29:29 N51:59 NXB MOV N29:30 N51:60 BND NXB MOV 1 N51:56 NXB MOV 4 N51:57 BND BND EOR
%   N51:8/13  "- HMI Input - Profile Edit Banding Open" %
%   N51:56  "- HMI Input - Profile Edit Band Display" %
%   N51:57  "- HMI Input - Profile Edit Band Number" %
%   N51:58  "- HMI Input - Profile Edit Band Reference" %
%   N29:22  "HMI Input Profile Band 1 Reference" %
%   N29:25  "HMI Input Profile Band 2 Reference" %
%   N29:28  "HMI Input Profile Band 3 Reference" %
%   N29:31  "HMI Input Profile Band 4 Reference" %
%   N51:59  "- HMI Input - Profile Edit Band Location" %
%   N29:20  "HMI Input Profile Band 1 Location" %
%   N29:23  "HMI Input Profile Band 2 Location" %
%   N29:26  "HMI Input Profile Band 3 Location" %
%   N29:29  "HMI Input Profile Band 4 Location" %
%   N51:60  "- HMI Input - Profile Edit Band Wraps" %
%   N29:21  "HMI Input Profile Band 1 Wraps" %
%   N29:24  "HMI Input Profile Band 2 Wraps" %
%   N29:27  "HMI Input Profile Band 3 Wraps" %
%   N29:30  "HMI Input Profile Band 4 Wraps" %
%   B3:7/1  "Profile Edit Band Reference Oneshot" %

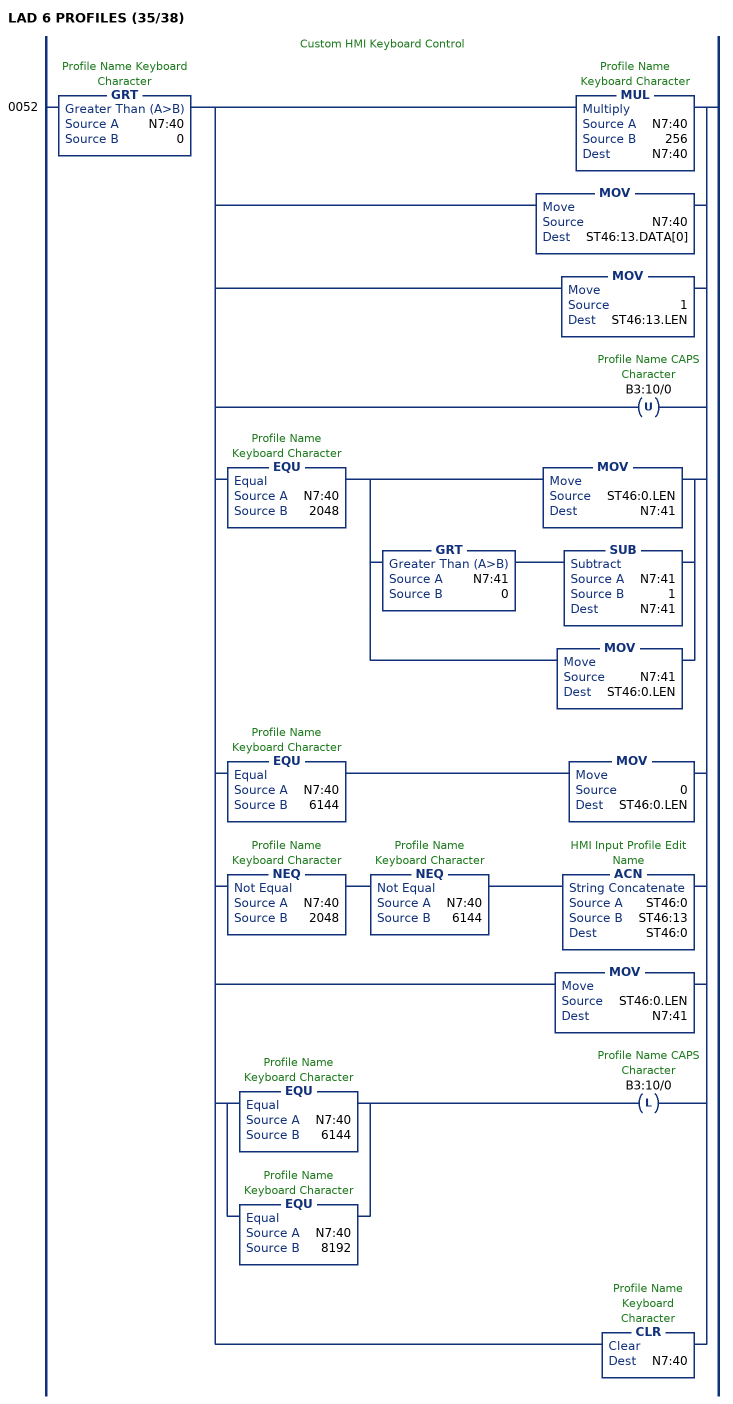
% Rung: 52 %
% Custom HMI Keyboard Control %
SOR GRT N7:40 0 BST MUL N7:40 256 N7:40 NXB BST MOV N7:40 ST46:13.DATA[0] NXB MOV 1 ST46:13.LEN BND NXB OTU B3:10/0 NXB EQU N7:40 2048 BST MOV ST46:0.LEN N7:41 NXB GRT N7:41 0 SUB N7:41 1 N7:41 NXB MOV N7:41 ST46:0.LEN BND NXB EQU N7:40 6144 MOV 0 ST46:0.LEN NXB NEQ N7:40 2048 NEQ N7:40 6144 ACN ST46:0 ST46:13 ST46:0 NXB MOV ST46:0.LEN N7:41 NXB BST EQU N7:40 6144 NXB EQU N7:40 8192 BND OTL B3:10/0 NXB CLR N7:40 BND EOR
%   N7:40  "Profile Name Keyboard Character" %
%   B3:10/0  "Profile Name CAPS Character" %
%   ST46:0  "HMI Input Profile Edit Name" %

